{attribute addProperty BoxType "EL3773-0000-0016"}
{attribute addProperty Id "I1_SAMPLESAT %I*ARRAY [1..10] OF INT16020"}
{attribute addProperty CRC "2535542409"}
{attribute addProperty SizeInBites "160"}
{attribute addProperty SizeInBytes "20"}
TYPE L1_Current_Samples_97214E89 :
STRUCT
	{attribute addProperty Name "I1_SAMPLES"}
	I1_SAMPLES AT %I* : ARRAY [1..10] OF INT;
END_STRUCT
END_TYPE

(* stored: Version 1.2.0.0, ProductVersion 3.1.4024.9
   DUT L1_Current_Samples_97214E89: Id {98137e46-e954-4df0-9aa1-9137f2b5ed2d} *)
